TYPE ST_MachineRecipe :
	STRUCT
	END_STRUCT
END_TYPE

(* stored: Version 1.1.0.1, ProductVersion 3.1.4024.12
   DUT ST_MachineRecipe: Id {07d75730-416c-41da-92b5-fede231f0a1e} *)
